{attribute 'enable_dynamic_creation'}
FUNCTION_BLOCK Track IMPLEMENTS ITF_Cyclic, ITF_Track
VAR
	MyTrackLength : LREAL;
END_VAR

{warning 'add method implementation '}
METHOD Cycle : BOOL
END_METHOD

METHOD Length : bool
VAR_INPUT
	TrackLength : LREAL;
END_VAR
MyTrackLength := TrackLength;
END_METHOD

END_FUNCTION_BLOCK

(* stored: Version 1.1.0.1, ProductVersion 3.1.4024.12
   POU Track: Id {85367b14-735c-4b56-a6a4-1e4f0d6b84de}, SpecialFunc None
   Method Cycle: Id {143b5232-be14-4dd2-a974-cabdb0e0e60e}
   Method Length: Id {c9f58fce-3361-4d24-95f8-0006eb3175ad} *)
